FUNCTION_BLOCK PUBLIC FB_DecoratorSalami EXTENDS FB_Decorator
VAR_INPUT
END_VAR
VAR_OUTPUT
END_VAR
VAR
END_VAR

METHOD GetDescription : STRING
IF (SUPER^.ipSideOrder <> 0) THEN
	GetDescription := CONCAT (SUPER^.ipSideOrder.GetDescription(), ' - Salami');
END_IF
END_METHOD

METHOD GetPrice : LREAL
IF (SUPER^.ipSideOrder <> 0) THEN
	GetPrice := SUPER^.ipSideOrder.GetPrice() + 1.4;
END_IF
END_METHOD

END_FUNCTION_BLOCK

(* stored: Version 1.1.0.1, ProductVersion 3.1.4022.16
   POU FB_DecoratorSalami: Id {6d62391a-f1ad-4b41-af6e-12267a1c0c1a}, SpecialFunc None
   Method GetDescription: Id {399edfb9-0cc8-456a-9308-bf7a7f21fd39}
   Method GetPrice: Id {7ebac5b8-38c0-40da-95fe-41daf1fd174a} *)
